// TIA Portal V20 export
TYPE "typeSafetySensor"
// stored: Access Published, IsFailsafeCompliant true, Namespace Safety
   STRUCT
      UnwinderLeftCartDetectSensor : Bool;   // Unwinder Left Cart Detect Sensor
      UnwinderRightCartDetectSensor : Bool;   // Unwinder Right Cart Detect Sensor
      CoverDetectSensor : Bool;   // Cover Detect Sensor
   END_STRUCT;
END_TYPE
